PROGRAM Main
VAR
	f : RollingFile;	

	file_name : T_MaxString := 'C:\Logs\test.txt';
	open_file : BOOL;
	close_file : BOOL;
	line_to_write : T_MaxString := 'Gday cobber$L';
	write_line : BOOL;
	
	////////////////////////////////////////////////////////////////////////////////	

	core_logger : TcLogCore(BufferSize := 50 * 50 * (Tc2_System.MAX_STRING_LENGTH + Constants.FifoOverhead));
	logger : TcLog;
	ads_adapter : AdsLogTargetAdapter;
	file_adapter : FileLogTargetAdapter;
	
	trigger_log : BOOL;
	
	////////////////////////////////////////////////////////////////////////////////
	
	within_string : T_MaxString := 'this.is.a.test.log';
	found_index : INT;
	extension : T_MaxString;
	
	dev_id : DeviceIdentification;
	line : T_maxString;
END_VAR

IF open_file THEN
	f.Open(file_name, FileOpenMode.Append OR FileOpenMode.Text);
	
	IF f.IsOpen THEN
		open_file := FALSE;
	ELSIF f.IsErrored THEN
		open_file := FALSE;
	END_IF
END_IF

IF close_file THEN
	f.Close();
	
	IF f.IsClosed THEN
		close_file := FALSE;
	END_IF
END_IF

IF write_line THEN
	f.WriteString(line_to_write);
// 	IF  THEN
// 		write_line := FALSE;
// 	END_IF
END_IF

////////////////////////////////////////////////////////////////////////////////

found_index := FindLastOccurrence(within_string, '.');
extension := GetFileExtension(within_string);

dev_id.Initialise();

////////////////////////////////////////////////////////////////////////////////

core_logger
	.IncludeInstancePath()
	.MinimumLevel(LogLevel.Debug)
	.AddAdapter1(ads_adapter)
	.AddAdapter2(file_adapter
		.FilePath('C:\Users\User\workspaces\TcLog\logs')
		.FileName('tclog_sandbox.log')
		.SetRollingInterval(RollingInterval.Hourly)
		.DeleteLogFilesAfterDays(1))
	.RunLogger();

IF trigger_log THEN
	trigger_log := FALSE;
	logger.Debug('Yo');
END_IF

END_PROGRAM

(* stored: Version 1.1.0.1
   POU Main: Id {cd559602-e31e-4d5b-ae62-cc768a3b78df}, SpecialFunc None *)
